# EPICS autosave request: ADApp/Db/NDStdArrays_settings.req
$(P)$(A)PostImages
$(P)$(A)MinImageUpdate
$(P)$(A)BlockingCallbacks
